// Mitsubishi GX Works2 project: Production Line1   PLC: Q03UDV
// PLC_Program

// global labels: Line1
VAR_GLOBAL
  Start1_Man AT X0 : BOOL;
  Start1_Rem AT X1 : BOOL;
  Stop1_Man AT X2 : BOOL;
  Stop1_Rem AT X3 : BOOL;
  Line1_Run_Stat AT M0 : BOOL;
  Line1_Error_Stat AT M1 : BOOL;
  Lid1_Raw_In AT M2 : BOOL;
  Lid1_Conv1 AT Y0 : BOOL;
  Lid1_Conv2 AT Y1 : BOOL;
  Lid1_Conv3 AT Y2 : BOOL;
  Lid1_Sen1 AT X4 : BOOL;
  LMach1_Start_Timer AT T0 : TIMER;
  LMach1_Start AT X5 : BOOL;
  Lid1_Sen2 AT X6 : BOOL;
  LArm1_isBusy AT X7 : BOOL;
  Lid1_Conv4 AT Y3 : BOOL;
  Base1_Raw_In AT M12 : BOOL;
  Base1_Conv1 AT Y10 : BOOL;
  Base1_Conv2 AT Y11 : BOOL;
  Base1_Conv3 AT Y12 : BOOL;
  Base1_Sen1 AT X14 : BOOL;
  BMach1_Start_Timer AT T10 : TIMER;
  BMach1_Start AT X15 : BOOL;
  Base1_Sen2 AT X16 : BOOL;
  BArm1_isBusy AT X17 : BOOL;
  Base1_Conv4 AT Y13 : BOOL;
  Lid1_Conv5 AT Y4 : BOOL;
  Base1_Conv5 AT Y14 : BOOL;
  Lid1_Sen3 AT X8 : BOOL;
  Base1_Sen3 AT X18 : BOOL;
  Assem1_Wait AT T1 : TIMER;
  Assem1_Cont AT M3 : BOOL;
  Assem1_Trig AT M4 : BOOL;
  Assem1_Hold AT M5 : BOOL;
  Assem1_Z AT Y5 : BOOL;
  Assem1_Grab AT Y6 : BOOL;
  Assem1_X AT Y7 : BOOL;
  Assem1_Back AT M6 : BOOL;
  PAssem1_Hold AT M7 : BOOL;
  PAssem1_Trig AT M8 : BOOL;
  PAssem1_Conv1 AT Y8 : BOOL;
  PAssem1_Conv2 AT Y9 : BOOL;
  PAssem1_Vis AT X9 : BOOL;
  Base1_Clamp AT Y15 : BOOL;
  Lid1_Clamp AT Y16 : BOOL;
  Clamp1_Raise AT Y17 : BOOL;
  Lid1_Conv6 AT Y18 : BOOL;
  Base1_Conv6 AT Y19 : BOOL;
  Lid1_Sen4 AT X19 : BOOL;
  Base1_Sen4 AT X20 : BOOL;
  Base1_Vis1 AT X21 : BOOL;
  Lid1_Vis1 AT X22 : BOOL;
  Lid1_Turn AT Y20 : BOOL;
  Base1_Turn AT Y21 : BOOL;
  Lid1_Turn_Conv AT Y22 : BOOL;
  Base1_Turn_Conv AT Y23 : BOOL;
  PAssem1_Sen1 AT X23 : BOOL;
  PAssem1_Conv3 AT Y24 : BOOL;
  OK1_Sen AT X24 : BOOL;
  Pusher1 AT Y25 : BOOL;
  Lid1_Raw_Sen AT X25 : BOOL;
  Base1_Raw_Sen AT X26 : BOOL;
  PAssem1_Sen2 AT X27 : BOOL;
  Blue_Hold AT M9 : BOOL;
  Sort_Sen_Bool0 AT X28 : BOOL;
  Sort_Sen_Bool1 AT X29 : BOOL;
  Sort_Sen_Bool2 AT X30 : BOOL;
  Green_Hold AT M10 : BOOL;
  Stop_Blade AT Y26 : BOOL;
  Sort_X AT Y27 : BOOL;
  Sort_Z AT Y28 : BOOL;
  Sort_Grab AT Y29 : BOOL;
  Sort_Rotate AT Y30 : BOOL;
  Sort_Clamp AT Y31 : BOOL;
END_VAR

// global labels: Line2
VAR_GLOBAL
  Start_L2_Manual AT X2 : BOOL;
  Start_L2_Online AT X3 : BOOL;
  Stop_L2_Manual AT X2 : BOOL;
  Stop_L2_Online AT X3 : BOOL;
END_VAR

// task Task_01 (event TRUE, interval 0, priority 31): Start_Stop_1
// task Task_02 (event TRUE, interval 0, priority 31): Mach1
// task Task_03 (event TRUE, interval 0, priority 31): ToAssem1
// task Task_04 (event TRUE, interval 0, priority 31): Assembly1
// task Task_05 (event TRUE, interval 0, priority 31): 
// task Task_06 (event TRUE, interval 0, priority 31): ToQC1
// task SortProd (event TRUE, interval 0, priority 31): SortProd

PROGRAM Start_Stop_1
VAR
  conveyor : BOOL;
END_VAR
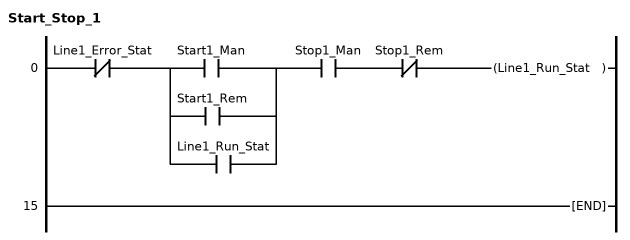
0     LDI     Line1_Error_Stat
      LD      Start1_Man
      OR      Start1_Rem
      OR      Line1_Run_Stat
      ANB
      AND     Stop1_Man
      ANI     Stop1_Rem
      OUT     Line1_Run_Stat
15    END
END_PROGRAM

PROGRAM Mach1
VAR
  Raw_In_1 : Raw_In;
  Lid_Raw_In : Raw_In;
  Base_Raw_In : Raw_In;
  Pre_Arm_Base1 : Pre_Arm;
  Pre_Arm_Base : Pre_Arm;
  Pre_Arm_Lid : Pre_Arm;
END_VAR
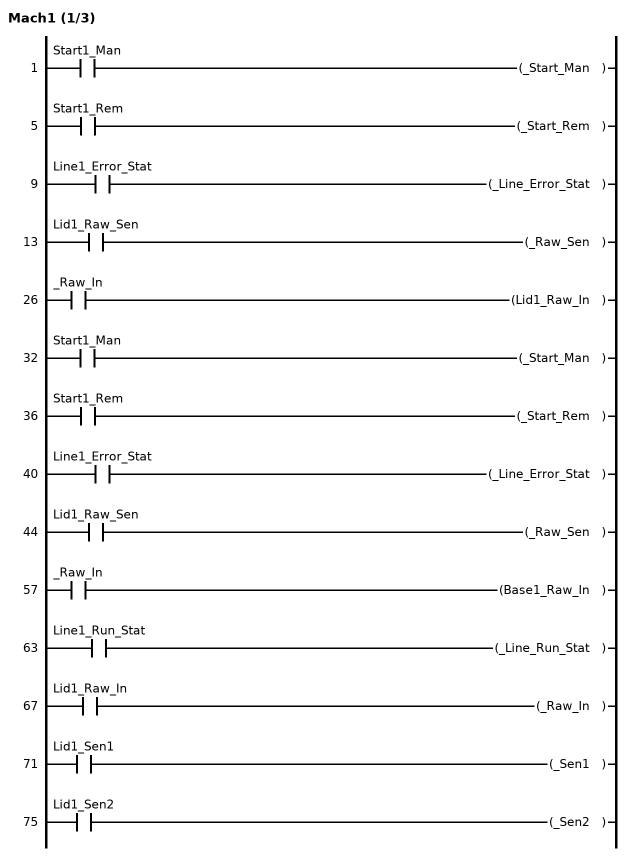
; FB BLK START Raw_In(Lid_Raw_In)
1     LD      Start1_Man
      OUT     _Start_Man
5     LD      Start1_Rem
      OUT     _Start_Rem
9     LD      Line1_Error_Stat
      OUT     _Line_Error_Stat
13    LD      Lid1_Raw_Sen
      OUT     _Raw_Sen
; FB START
; FB_NAME Raw_In
; INSTANCE_NAME Lid_Raw_In
; FB IN_B:Start_Man
; FB OUT_Raw_In:B
; FB IN_B:Start_Rem
; FB IN_B:Line_Error_Stat
; FB IN_B:Raw_Sen
; FB END
26    LD      _Raw_In
      OUT     Lid1_Raw_In
; FB BLK END
; FB BLK START Raw_In(Base_Raw_In)
32    LD      Start1_Man
      OUT     _Start_Man
36    LD      Start1_Rem
      OUT     _Start_Rem
40    LD      Line1_Error_Stat
      OUT     _Line_Error_Stat
44    LD      Lid1_Raw_Sen
      OUT     _Raw_Sen
; FB START
; FB_NAME Raw_In
; INSTANCE_NAME Base_Raw_In
; FB IN_B:Start_Man
; FB OUT_Raw_In:B
; FB IN_B:Start_Rem
; FB IN_B:Line_Error_Stat
; FB IN_B:Raw_Sen
; FB END
57    LD      _Raw_In
      OUT     Base1_Raw_In
; FB BLK END
; FB BLK START Pre_Arm(Pre_Arm_Lid)
63    LD      Line1_Run_Stat
      OUT     _Line_Run_Stat
67    LD      Lid1_Raw_In
      OUT     _Raw_In
71    LD      Lid1_Sen1
      OUT     _Sen1
75    LD      Lid1_Sen2
      OUT     _Sen2
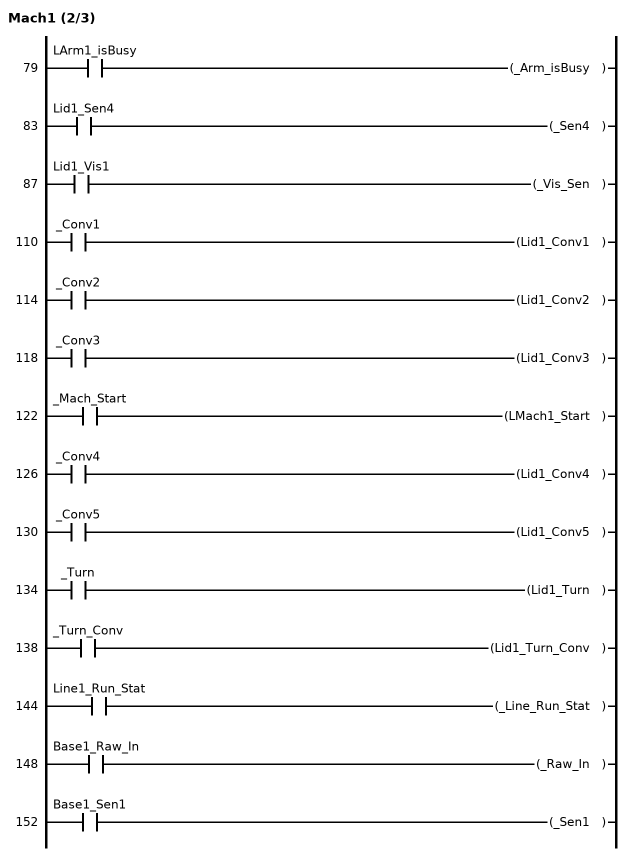
79    LD      LArm1_isBusy
      OUT     _Arm_isBusy
83    LD      Lid1_Sen4
      OUT     _Sen4
87    LD      Lid1_Vis1
      OUT     _Vis_Sen
; FB START
; FB_NAME Pre_Arm
; INSTANCE_NAME Pre_Arm_Lid
; FB IN_B:Line_Run_Stat
; FB OUT_Conv1:B
; FB IN_B:Raw_In
; FB OUT_Conv2:B
; FB IN_B:Sen1
; FB OUT_Conv3:B
; FB IN_B:Sen2
; FB OUT_Mach_Start:B
; FB IN_B:Arm_isBusy
; FB OUT_Conv4:B
; FB IN_B:Sen4
; FB OUT_Conv5:B
; FB IN_B:Vis_Sen
; FB OUT_Turn:B
; FB OUT_Turn_Conv:B
; FB END
110   LD      _Conv1
      OUT     Lid1_Conv1
114   LD      _Conv2
      OUT     Lid1_Conv2
118   LD      _Conv3
      OUT     Lid1_Conv3
122   LD      _Mach_Start
      OUT     LMach1_Start
126   LD      _Conv4
      OUT     Lid1_Conv4
130   LD      _Conv5
      OUT     Lid1_Conv5
134   LD      _Turn
      OUT     Lid1_Turn
138   LD      _Turn_Conv
      OUT     Lid1_Turn_Conv
; FB BLK END
; FB BLK START Pre_Arm(Pre_Arm_Base)
144   LD      Line1_Run_Stat
      OUT     _Line_Run_Stat
148   LD      Base1_Raw_In
      OUT     _Raw_In
152   LD      Base1_Sen1
      OUT     _Sen1
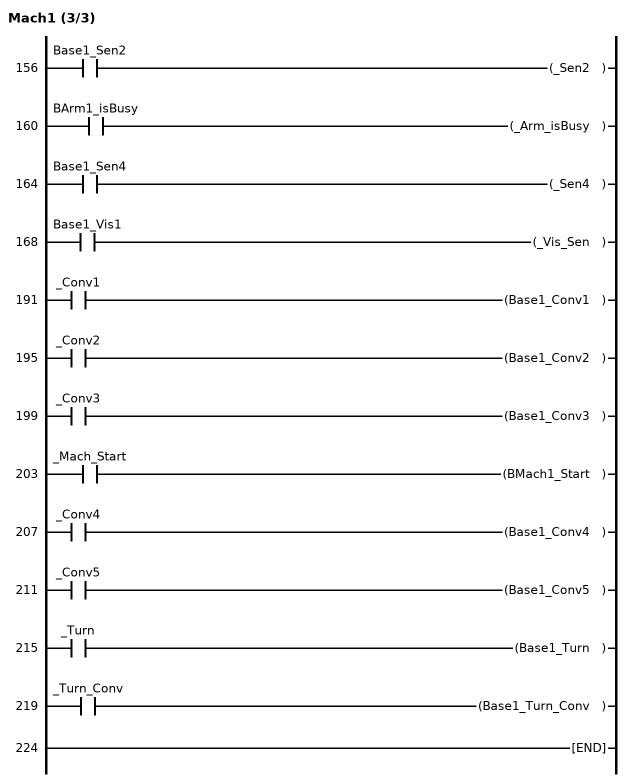
156   LD      Base1_Sen2
      OUT     _Sen2
160   LD      BArm1_isBusy
      OUT     _Arm_isBusy
164   LD      Base1_Sen4
      OUT     _Sen4
168   LD      Base1_Vis1
      OUT     _Vis_Sen
; FB START
; FB_NAME Pre_Arm
; INSTANCE_NAME Pre_Arm_Base
; FB IN_B:Line_Run_Stat
; FB OUT_Conv1:B
; FB IN_B:Raw_In
; FB OUT_Conv2:B
; FB IN_B:Sen1
; FB OUT_Conv3:B
; FB IN_B:Sen2
; FB OUT_Mach_Start:B
; FB IN_B:Arm_isBusy
; FB OUT_Conv4:B
; FB IN_B:Sen4
; FB OUT_Conv5:B
; FB IN_B:Vis_Sen
; FB OUT_Turn:B
; FB OUT_Turn_Conv:B
; FB END
191   LD      _Conv1
      OUT     Base1_Conv1
195   LD      _Conv2
      OUT     Base1_Conv2
199   LD      _Conv3
      OUT     Base1_Conv3
203   LD      _Mach_Start
      OUT     BMach1_Start
207   LD      _Conv4
      OUT     Base1_Conv4
211   LD      _Conv5
      OUT     Base1_Conv5
215   LD      _Turn
      OUT     Base1_Turn
219   LD      _Turn_Conv
      OUT     Base1_Turn_Conv
; FB BLK END
224   END
END_PROGRAM

PROGRAM ToAssem1
VAR
  Lid_Assem_Conv : Assem_Conv;
  Base_Assem_Conv : Assem_Conv;
  Post_Assem : Post_Assem;
END_VAR
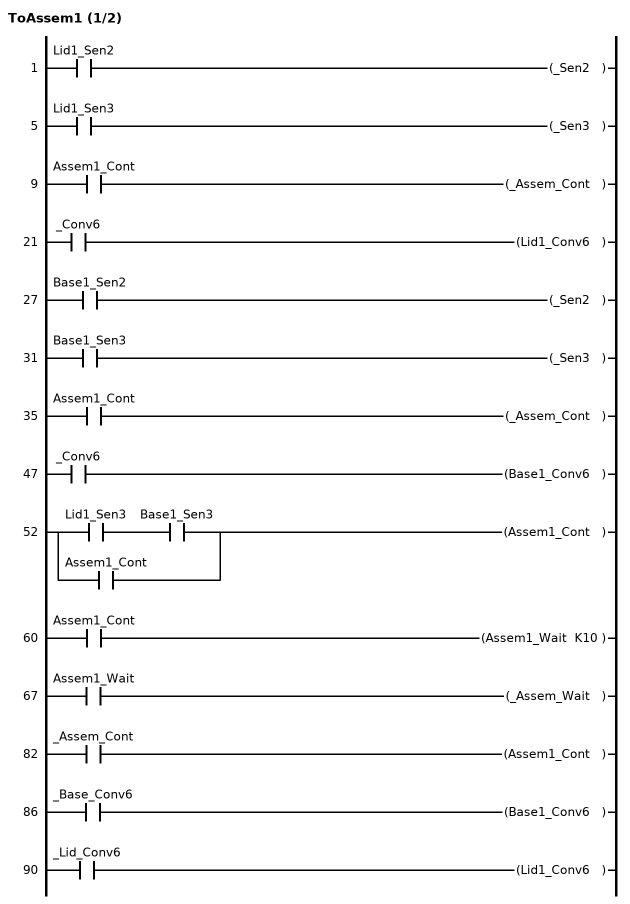
; FB BLK START Assem_Conv(Lid_Assem_Conv)
1     LD      Lid1_Sen2
      OUT     _Sen2
5     LD      Lid1_Sen3
      OUT     _Sen3
9     LD      Assem1_Cont
      OUT     _Assem_Cont
; FB START
; FB_NAME Assem_Conv
; INSTANCE_NAME Lid_Assem_Conv
; FB IN_B:Sen2
; FB OUT_Conv6:B
; FB IN_B:Sen3
; FB IN_B:Assem_Cont
; FB END
21    LD      _Conv6
      OUT     Lid1_Conv6
; FB BLK END
; FB BLK START Assem_Conv(Base_Assem_Conv)
27    LD      Base1_Sen2
      OUT     _Sen2
31    LD      Base1_Sen3
      OUT     _Sen3
35    LD      Assem1_Cont
      OUT     _Assem_Cont
; FB START
; FB_NAME Assem_Conv
; INSTANCE_NAME Base_Assem_Conv
; FB IN_B:Sen2
; FB OUT_Conv6:B
; FB IN_B:Sen3
; FB IN_B:Assem_Cont
; FB END
47    LD      _Conv6
      OUT     Base1_Conv6
; FB BLK END
52    LD      Lid1_Sen3
      AND     Base1_Sen3
      OR      Assem1_Cont
      OUT     Assem1_Cont
60    LD      Assem1_Cont
      OUT     Assem1_Wait K10
; FB BLK START Post_Assem(Post_Assem)
67    LD      Assem1_Wait
      OUT     _Assem_Wait
; FB START
; FB_NAME Post_Assem
; INSTANCE_NAME Post_Assem
; FB IN_B:Assem_Wait
; FB OUT_Assem_Cont:B
; FB OUT_Base_Conv6:B
; FB OUT_Lid_Conv6:B
; FB OUT_Assem_Trig:B
; FB OUT_Base_Clamp:B
; FB OUT_Lid_Clamp:B
; FB END
82    LD      _Assem_Cont
      OUT     Assem1_Cont
86    LD      _Base_Conv6
      OUT     Base1_Conv6
90    LD      _Lid_Conv6
      OUT     Lid1_Conv6
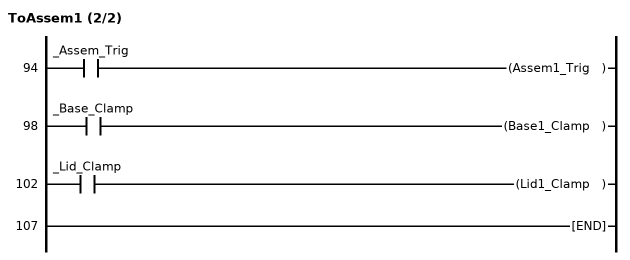
94    LD      _Assem_Trig
      OUT     Assem1_Trig
98    LD      _Base_Clamp
      OUT     Base1_Clamp
102   LD      _Lid_Clamp
      OUT     Lid1_Clamp
; FB BLK END
107   END
END_PROGRAM

PROGRAM Assembly1
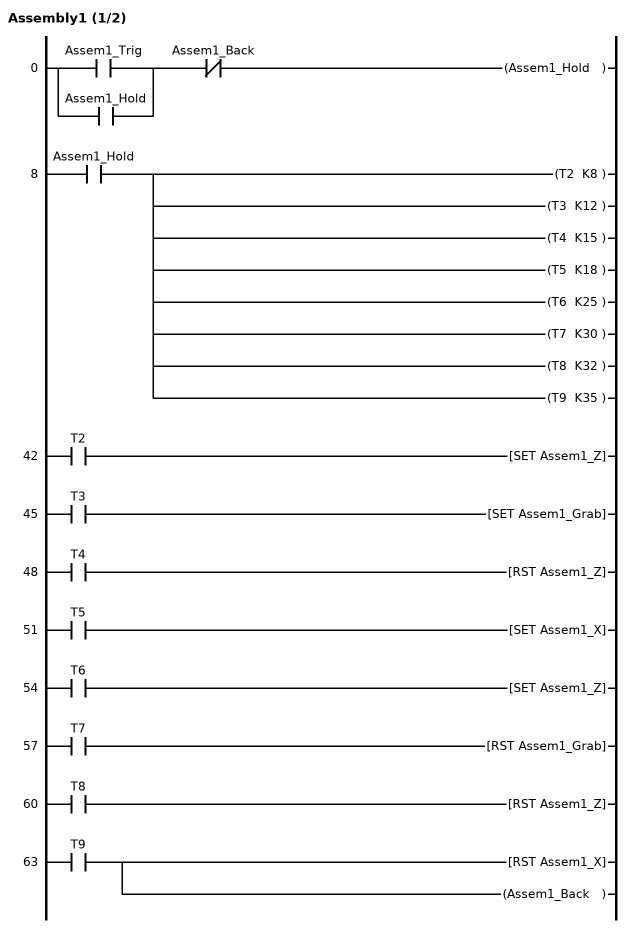
0     LD      Assem1_Trig
      OR      Assem1_Hold
      ANI     Assem1_Back
      OUT     Assem1_Hold
8     LD      Assem1_Hold
      OUT     T2 K8
      OUT     T3 K12
      OUT     T4 K15
      OUT     T5 K18
      OUT     T6 K25
      OUT     T7 K30
      OUT     T8 K32
      OUT     T9 K35
42    LD      T2
      SET     Assem1_Z
45    LD      T3
      SET     Assem1_Grab
48    LD      T4
      RST     Assem1_Z
51    LD      T5
      SET     Assem1_X
54    LD      T6
      SET     Assem1_Z
57    LD      T7
      RST     Assem1_Grab
60    LD      T8
      RST     Assem1_Z
63    LD      T9
      RST     Assem1_X
      OUT     Assem1_Back
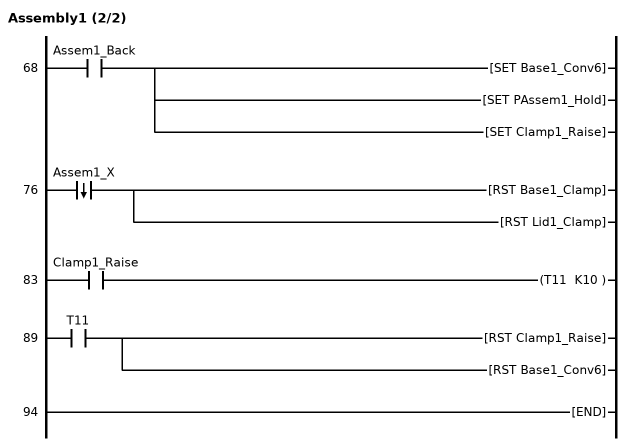
68    LD      Assem1_Back
      SET     Base1_Conv6
      SET     PAssem1_Hold
      SET     Clamp1_Raise
76    LDF     Assem1_X
      RST     Base1_Clamp
      RST     Lid1_Clamp
83    LD      Clamp1_Raise
      OUT     T11 K10
89    LD      T11
      RST     Clamp1_Raise
      RST     Base1_Conv6
94    END
END_PROGRAM

FUNCTION_BLOCK Raw_In
VAR_INPUT
  Start_Man : BOOL;
  Start_Rem : BOOL;
END_VAR
VAR_OUTPUT
  Raw_In : BOOL;
END_VAR
VAR_INPUT
  Line_Error_Stat : BOOL;
  Raw_Sen : BOOL;
END_VAR
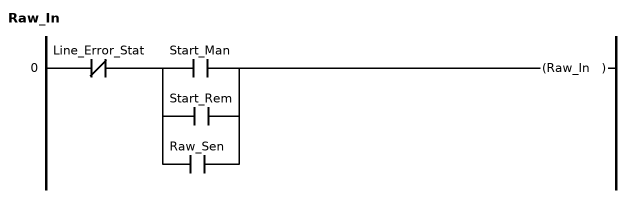
0     LDI     Line_Error_Stat
      LD      Start_Man
      OR      Start_Rem
      OR      Raw_Sen
      ANB
      OUT     Raw_In
END_FUNCTION_BLOCK

FUNCTION_BLOCK Pre_Arm
VAR_INPUT
  Line_Run_Stat : BOOL;
  Raw_In : BOOL;
END_VAR
VAR_OUTPUT
  Conv1 : BOOL;
  Conv2 : BOOL;
  Conv3 : BOOL;
END_VAR
VAR_INPUT
  Sen1 : BOOL;
  Sen2 : BOOL;
END_VAR
VAR
  Mach_Start_Timer : TIMER;
END_VAR
VAR_OUTPUT
  Mach_Start : BOOL;
  Conv4 : BOOL;
END_VAR
VAR_INPUT
  Arm_isBusy : BOOL;
END_VAR
VAR_OUTPUT
  Conv5 : BOOL;
END_VAR
VAR_INPUT
  Sen4 : BOOL;
END_VAR
VAR_OUTPUT
  Turn : BOOL;
END_VAR
VAR_INPUT
  Vis_Sen : BOOL;
END_VAR
VAR_OUTPUT
  Turn_Conv : BOOL;
END_VAR
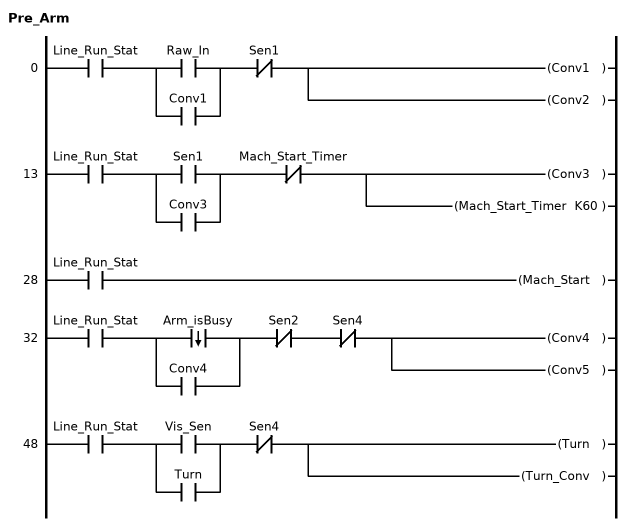
0     LD      Line_Run_Stat
      LD      Raw_In
      OR      Conv1
      ANB
      ANI     Sen1
      OUT     Conv1
      OUT     Conv2
13    LD      Line_Run_Stat
      LD      Sen1
      OR      Conv3
      ANB
      ANI     Mach_Start_Timer
      OUT     Conv3
      OUT     Mach_Start_Timer K60
28    LD      Line_Run_Stat
      OUT     Mach_Start
32    LD      Line_Run_Stat
      LDF     Arm_isBusy
      OR      Conv4
      ANB
      ANI     Sen2
      ANI     Sen4
      OUT     Conv4
      OUT     Conv5
48    LD      Line_Run_Stat
      LD      Vis_Sen
      OR      Turn
      ANB
      ANI     Sen4
      OUT     Turn
      OUT     Turn_Conv
END_FUNCTION_BLOCK

PROGRAM ToQC1
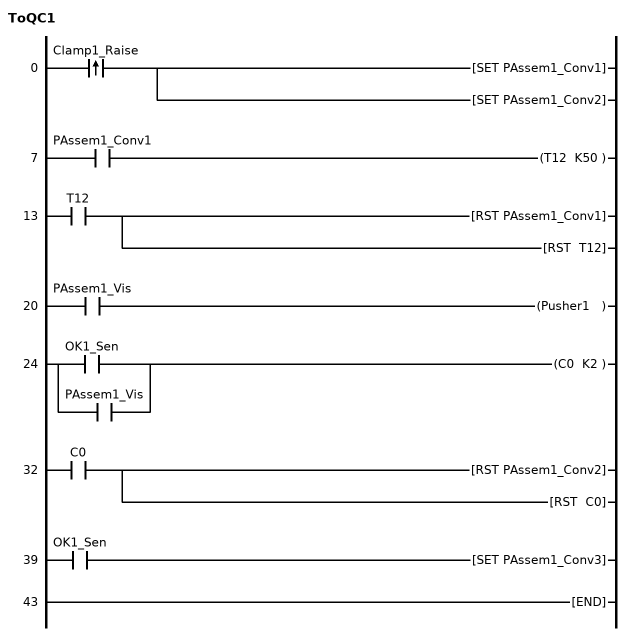
0     LDP     Clamp1_Raise
      SET     PAssem1_Conv1
      SET     PAssem1_Conv2
7     LD      PAssem1_Conv1
      OUT     T12 K50
13    LD      T12
      RST     PAssem1_Conv1
      RST     T12
20    LD      PAssem1_Vis
      OUT     Pusher1
24    LD      OK1_Sen
      OR      PAssem1_Vis
      OUT     C0 K2
32    LD      C0
      RST     PAssem1_Conv2
      RST     C0
39    LD      OK1_Sen
      SET     PAssem1_Conv3
43    END
END_PROGRAM

FUNCTION_BLOCK Assem_Conv
VAR_INPUT
  Sen2 : BOOL;
  Sen3 : BOOL;
END_VAR
VAR_OUTPUT
  Conv6 : BOOL;
END_VAR
VAR_INPUT
  Assem_Cont : BOOL;
END_VAR
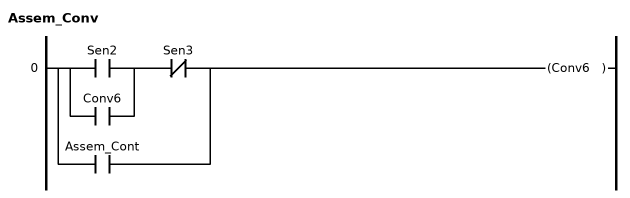
0     LD      Sen2
      OR      Conv6
      ANI     Sen3
      OR      Assem_Cont
      OUT     Conv6
END_FUNCTION_BLOCK

FUNCTION_BLOCK Post_Assem
VAR_INPUT
  Assem_Wait : BOOL;
END_VAR
VAR_OUTPUT
  Assem_Cont : BOOL;
  Base_Conv6 : BOOL;
  Assem_Trig : BOOL;
  Base_Clamp : BOOL;
  Lid_Clamp : BOOL;
  Lid_Conv6 : BOOL;
END_VAR
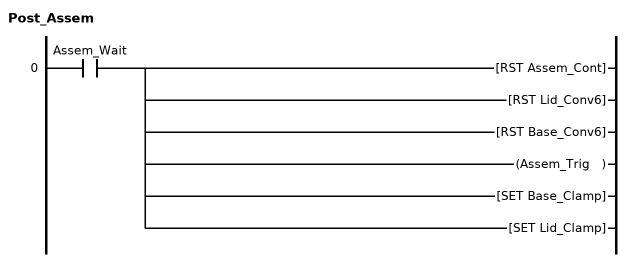
0     LD      Assem_Wait
      RST     Assem_Cont
      RST     Lid_Conv6
      RST     Base_Conv6
      OUT     Assem_Trig
      SET     Base_Clamp
      SET     Lid_Clamp
END_FUNCTION_BLOCK

PROGRAM SortProd
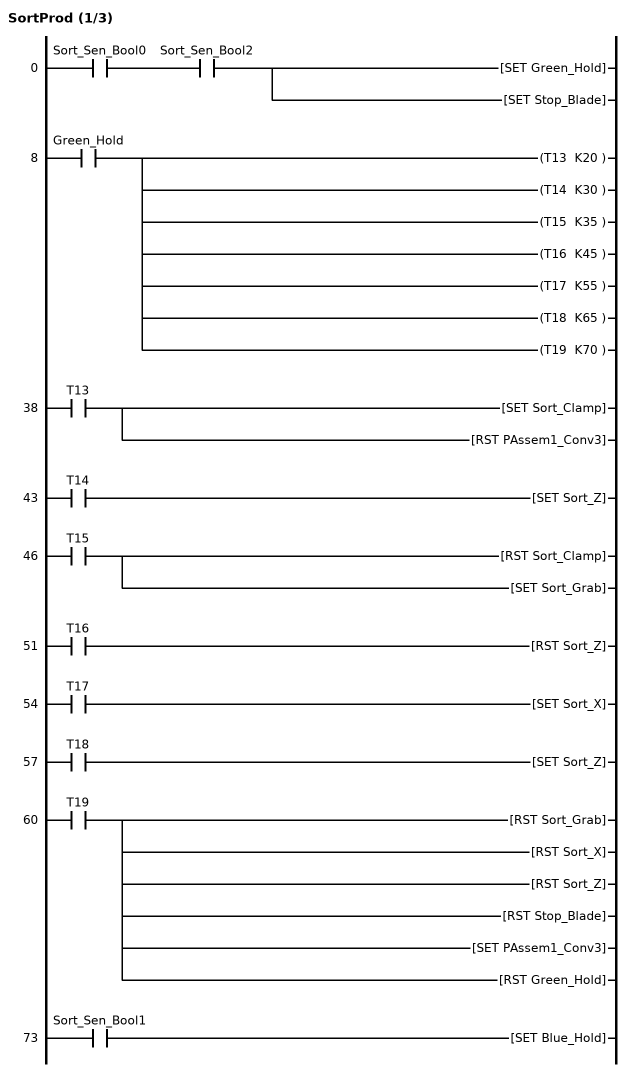
0     LD      Sort_Sen_Bool0
      AND     Sort_Sen_Bool2
      SET     Green_Hold
      SET     Stop_Blade
8     LD      Green_Hold
      OUT     T13 K20
      OUT     T14 K30
      OUT     T15 K35
      OUT     T16 K45
      OUT     T17 K55
      OUT     T18 K65
      OUT     T19 K70
38    LD      T13
      SET     Sort_Clamp
      RST     PAssem1_Conv3
43    LD      T14
      SET     Sort_Z
46    LD      T15
      RST     Sort_Clamp
      SET     Sort_Grab
51    LD      T16
      RST     Sort_Z
54    LD      T17
      SET     Sort_X
57    LD      T18
      SET     Sort_Z
60    LD      T19
      RST     Sort_Grab
      RST     Sort_X
      RST     Sort_Z
      RST     Stop_Blade
      SET     PAssem1_Conv3
      RST     Green_Hold
73    LD      Sort_Sen_Bool1
      SET     Blue_Hold
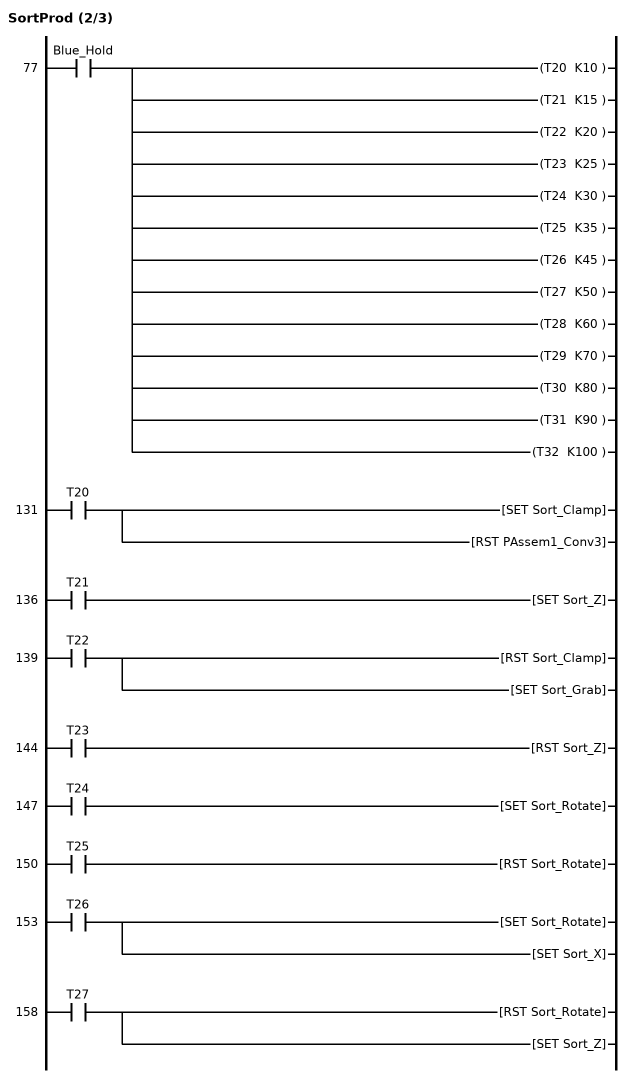
77    LD      Blue_Hold
      OUT     T20 K10
      OUT     T21 K15
      OUT     T22 K20
      OUT     T23 K25
      OUT     T24 K30
      OUT     T25 K35
      OUT     T26 K45
      OUT     T27 K50
      OUT     T28 K60
      OUT     T29 K70
      OUT     T30 K80
      OUT     T31 K90
      OUT     T32 K100
131   LD      T20
      SET     Sort_Clamp
      RST     PAssem1_Conv3
136   LD      T21
      SET     Sort_Z
139   LD      T22
      RST     Sort_Clamp
      SET     Sort_Grab
144   LD      T23
      RST     Sort_Z
147   LD      T24
      SET     Sort_Rotate
150   LD      T25
      RST     Sort_Rotate
153   LD      T26
      SET     Sort_Rotate
      SET     Sort_X
158   LD      T27
      RST     Sort_Rotate
      SET     Sort_Z
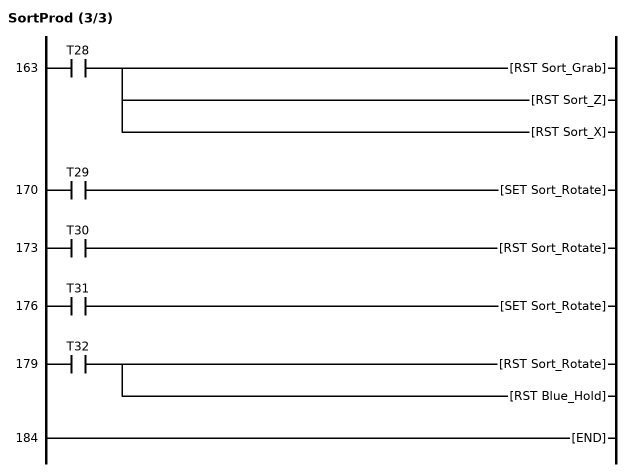
163   LD      T28
      RST     Sort_Grab
      RST     Sort_Z
      RST     Sort_X
170   LD      T29
      SET     Sort_Rotate
173   LD      T30
      RST     Sort_Rotate
176   LD      T31
      SET     Sort_Rotate
179   LD      T32
      RST     Sort_Rotate
      RST     Blue_Hold
184   END
END_PROGRAM
